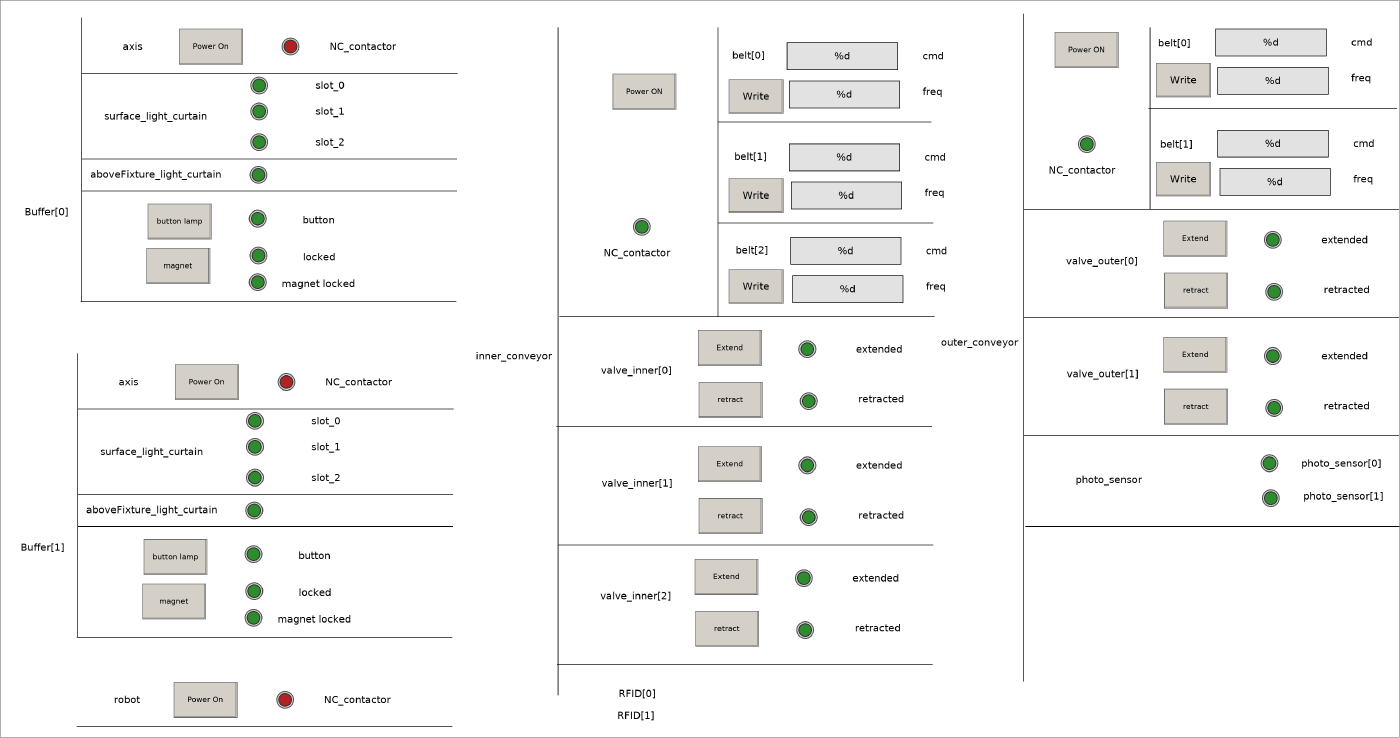
VISUALIZATION v_pm_0  // 2048x1080
VAR_IN_OUT
	dIO_PM		: Picking_Module;
END_VAR
    Lamp1 (364,110 30x30), variable: dIO_PM.buffer[0].surfae_slot_0, style: Lamp-Lamp1-Green
    Label (418,112 130x26), "slot_0"
    Label (28,297 80x26), "Buffer[0]"
    Line (120,107) (669,107)
    Line (119,26) (119,441)
    Line (118,441) (667,441)
    Label (672,508 160x26), "inner_conveyor"
    Line (816,40) (816,1017)
    Label (851,529 160x26), "valve_inner[0]"
    Button (1021,483 93x52), "Extend", colour toggle: dIO_PM.inConv.valve[0].extend
        OnMouseDown: execute { dIO_PM.inConv.valve[0].extend := TRUE; dIO_PM.inConv.valve[0].retract := FALSE; }
    Button (1022,559 93x52), "retract", colour toggle: dIO_PM.inConv.valve[0].retract
        OnMouseDown: execute { dIO_PM.inConv.valve[0].extend := FALSE; dIO_PM.inConv.valve[0].retract := TRUE; }
    Lamp1 (1166,496 30x30), variable: dIO_PM.inConv.valve[0].extended, style: Lamp-Lamp1-Green
    Lamp1 (1168,572 30x30), variable: dIO_PM.inConv.valve[0].retracted, style: Lamp-Lamp1-Green
    Label (1220,498 132x26), "extended"
    Label (1223,571 132x26), "retracted"
    Label (852,694 160x26), "valve_inner[1]"
    Label (850,859 160x26), "valve_inner[2]"
    Line (814,624) (1363,624)
    Line (816,797) (1365,797)
    Line (815,972) (1364,972)
    Label (465,55 132x26), "NC_contactor"
    Label (128,55 132x26), "axis"
    Button (262,42 93x52), "Power On", colour toggle: dIO_PM.buffer[0].power_axis
        toggle dIO_PM.buffer[0].power_axis
    Lamp1 (410,53 30x30), variable: dIO_PM.buffer[0].contractor_axis, style: Lamp-Lamp1-Red
    Label (128,157 200x26), "surface_light_curtain"
    Label (418,150 130x26), "slot_1"
    Lamp1 (364,148 30x30), variable: dIO_PM.buffer[0].surfae_slot_1, style: Lamp-Lamp1-Green
    Label (418,195 130x26), "slot_2"
    Lamp1 (364,193 30x30), variable: dIO_PM.buffer[0].surfae_slot_2, style: Lamp-Lamp1-Green
    Label (128,242 200x26), "aboveFixture_light_curtain"
    Lamp1 (363,241 30x30), variable: dIO_PM.buffer[0].above_fixture_light_curtain, style: Lamp-Lamp1-Green
    Line (119,232) (668,232)
    Line (119,279) (668,279)
    Label (406,309 120x26), "button"
    Lamp1 (362,305 30x30), variable: dIO_PM.buffer[0].button, style: Lamp-Lamp1-Green
    Button (216,298 93x52), "button lamp", colour toggle: dIO_PM.buffer[0].lamp_button
        toggle dIO_PM.buffer[0].lamp_button
    Button (214,363 93x52), "magnet", colour toggle: dIO_PM.buffer[0].magnet
        toggle dIO_PM.buffer[0].magnet
    Label (407,363 120x26), "locked"
    Lamp1 (363,359 30x30), variable: dIO_PM.buffer[0].locked, style: Lamp-Lamp1-Green
    Label (406,402 120x26), "magnet locked"
    Lamp1 (362,398 30x30), variable: dIO_PM.buffer[0].magnet_locked, style: Lamp-Lamp1-Green
    Lamp1 (358,601 30x30), variable: dIO_PM.buffer[1].surfae_slot_0, style: Lamp-Lamp1-Green
    Label (412,603 130x26), "slot_0"
    Label (22,788 80x26), "Buffer[1]"
    Line (114,598) (663,598)
    Line (113,517) (113,932)
    Line (112,932) (661,932)
    Label (459,546 132x26), "NC_contactor"
    Label (122,546 132x26), "axis"
    Button (256,533 93x52), "Power On", colour toggle: dIO_PM.buffer[1].power_axis
        toggle dIO_PM.buffer[1].power_axis
    Lamp1 (404,544 30x30), variable: dIO_PM.buffer[1].contractor_axis, style: Lamp-Lamp1-Red
    Label (122,648 200x26), "surface_light_curtain"
    Label (412,641 130x26), "slot_1"
    Lamp1 (358,639 30x30), variable: dIO_PM.buffer[1].surfae_slot_1, style: Lamp-Lamp1-Green
    Label (412,686 130x26), "slot_2"
    Lamp1 (358,684 30x30), variable: dIO_PM.buffer[1].surfae_slot_2, style: Lamp-Lamp1-Green
    Label (122,733 200x26), "aboveFixture_light_curtain"
    Lamp1 (357,732 30x30), variable: dIO_PM.buffer[1].above_fixture_light_curtain, style: Lamp-Lamp1-Green
    Line (113,723) (662,723)
    Line (113,770) (662,770)
    Label (400,800 120x26), "button"
    Lamp1 (356,796 30x30), variable: dIO_PM.buffer[1].button, style: Lamp-Lamp1-Green
    Button (210,789 93x52), "button lamp", colour toggle: dIO_PM.buffer[1].lamp_button
        toggle dIO_PM.buffer[1].lamp_button
    Button (208,854 93x52), "magnet", colour toggle: dIO_PM.buffer[1].magnet
        toggle dIO_PM.buffer[1].magnet
    Label (401,854 120x26), "locked"
    Lamp1 (357,850 30x30), variable: dIO_PM.buffer[1].locked, style: Lamp-Lamp1-Green
    Label (400,893 120x26), "magnet locked"
    Lamp1 (356,889 30x30), variable: dIO_PM.buffer[1].magnet_locked, style: Lamp-Lamp1-Green
    Line (112,1063) (661,1063)
    Label (457,1011 132x26), "NC_contactor"
    Label (120,1011 132x26), "robot"
    Button (254,998 93x52), "Power On", colour toggle: dIO_PM.power_robot
        toggle dIO_PM.power_robot
    Lamp1 (402,1009 30x30), variable: dIO_PM.contactor_robot, style: Lamp-Lamp1-Red
    Rectangle (1151,62 162x40), "%d", text variable: dIO_PM.inConv.belt[0].fbconverter.cmd
        OnMouseClick: write the text variable via Default
    Rectangle (1154,118 162x40), "%d", text variable: dIO_PM.inConv.belt[0].fbconverter.freq
        OnMouseClick: write the text variable via Default
    Label (1029,68 132x26), "belt[0]"
    Label (1299,69 132x26), "cmd"
    Label (1298,121 132x26), "freq"
    Line (1050,178) (1362,178)
    Rectangle (1154,210 162x40), "%d", text variable: dIO_PM.inConv.belt[1].fbconverter.cmd
        OnMouseClick: write the text variable via Default
    Rectangle (1157,266 162x40), "%d", text variable: dIO_PM.inConv.belt[1].fbconverter.freq
        OnMouseClick: write the text variable via Default
    Label (1032,216 132x26), "belt[1]"
    Label (1302,217 132x26), "cmd"
    Label (1301,269 132x26), "freq"
    Line (1050,326) (1365,326)
    Rectangle (1156,347 162x40), "%d", text variable: dIO_PM.inConv.belt[2].fbconverter.cmd
        OnMouseClick: write the text variable via Default
    Rectangle (1159,403 162x40), "%d", text variable: dIO_PM.inConv.belt[2].fbconverter.freq
        OnMouseClick: write the text variable via Default
    Label (1034,353 132x26), "belt[2]"
    Label (1304,354 132x26), "cmd"
    Label (1303,406 132x26), "freq"
    Line (818,463) (1367,463)
    Button (1021,653 93x52), "Extend", colour toggle: dIO_PM.inConv.valve[1].extend
        OnMouseDown: execute { dIO_PM.inConv.valve[1].extend := TRUE; dIO_PM.inConv.valve[1].retract := FALSE; }
    Button (1022,729 93x52), "retract", colour toggle: dIO_PM.inConv.valve[1].retract
        OnMouseDown: execute { dIO_PM.inConv.valve[1].extend := FALSE; dIO_PM.inConv.valve[1].retract := TRUE; }
    Lamp1 (1166,666 30x30), variable: dIO_PM.inConv.valve[1].extended, style: Lamp-Lamp1-Green
    Lamp1 (1168,742 30x30), variable: dIO_PM.inConv.valve[1].retracted, style: Lamp-Lamp1-Green
    Label (1220,668 132x26), "extended"
    Label (1223,741 132x26), "retracted"
    Button (1016,818 93x52), "Extend", colour toggle: dIO_PM.inConv.valve[2].extend
        OnMouseDown: execute { dIO_PM.inConv.valve[2].extend := TRUE; dIO_PM.inConv.valve[2].retract := FALSE; }
    Button (1017,894 93x52), "retract", colour toggle: dIO_PM.inConv.valve[2].retract
        OnMouseDown: execute { dIO_PM.inConv.valve[2].extend := FALSE; dIO_PM.inConv.valve[2].retract := TRUE; }
    Lamp1 (1161,831 30x30), variable: dIO_PM.inConv.valve[2].extended, style: Lamp-Lamp1-Green
    Lamp1 (1163,907 30x30), variable: dIO_PM.inConv.valve[2].retracted, style: Lamp-Lamp1-Green
    Label (1215,833 132x26), "extended"
    Label (1218,906 132x26), "retracted"
    Label (852,1002 160x26), "RFID[0]"
    Label (850,1034 160x26), "RFID[1]"
    Label (1353,488 160x26), "outer_conveyor"
    Line (1497,20) (1497,997)
    Label (1532,369 160x26), "valve_outer[0]"
    Button (1702,323 93x52), "Extend", colour toggle: dIO_PM.outConv.valve[0].extend
        OnMouseDown: execute { dIO_PM.outConv.valve[0].extend := TRUE; dIO_PM.outConv.valve[0].retract := FALSE; }
    Button (1703,399 93x52), "retract", colour toggle: dIO_PM.outConv.valve[0].retract
        OnMouseDown: execute { dIO_PM.outConv.valve[0].extend := FALSE; dIO_PM.outConv.valve[0].retract := TRUE; }
    Lamp1 (1847,336 30x30), variable: dIO_PM.outConv.valve[0].extended, style: Lamp-Lamp1-Green
    Lamp1 (1849,412 30x30), variable: dIO_PM.outConv.valve[0].retracted, style: Lamp-Lamp1-Green
    Label (1901,338 132x26), "extended"
    Label (1904,411 132x26), "retracted"
    Label (1533,534 160x26), "valve_outer[1]"
    Line (1498,464) (2047,464)
    Line (1497,637) (2046,637)
    Line (1500,770) (2049,770)
    Rectangle (1778,42 162x40), "%d", text variable: dIO_PM.outConv.belt[0].fbconverter.cmd
        OnMouseClick: write the text variable via Default
    Rectangle (1781,98 162x40), "%d", text variable: dIO_PM.outConv.belt[0].fbconverter.freq
        OnMouseClick: write the text variable via Default
    Label (1652,50 132x26), "belt[0]"
    Label (1926,49 132x26), "cmd"
    Label (1925,101 132x26), "freq"
    Line (1680,158) (2043,158)
    Rectangle (1781,190 162x40), "%d", text variable: dIO_PM.outConv.belt[1].fbconverter.cmd
        OnMouseClick: write the text variable via Default
    Rectangle (1784,246 162x40), "%d", text variable: dIO_PM.outConv.belt[1].fbconverter.freq
        OnMouseClick: write the text variable via Default
    Label (1655,198 132x26), "belt[1]"
    Label (1929,197 132x26), "cmd"
    Label (1928,249 132x26), "freq"
    Line (1497,306) (2046,306)
    Button (1702,493 93x52), "Extend", colour toggle: dIO_PM.outConv.valve[1].extend
        OnMouseDown: execute { dIO_PM.outConv.valve[1].extend := TRUE; dIO_PM.outConv.valve[1].retract := FALSE; }
    Button (1703,569 93x52), "retract", colour toggle: dIO_PM.outConv.valve[1].retract
        OnMouseDown: execute { dIO_PM.outConv.valve[1].extend := FALSE; dIO_PM.outConv.valve[1].retract := TRUE; }
    Lamp1 (1847,506 30x30), variable: dIO_PM.outConv.valve[1].extended, style: Lamp-Lamp1-Green
    Lamp1 (1849,582 30x30), variable: dIO_PM.outConv.valve[1].retracted, style: Lamp-Lamp1-Green
    Label (1901,508 132x26), "extended"
    Label (1904,581 132x26), "retracted"
    Lamp1 (1842,663 30x30), variable: dIO_PM.outConv.photo_sensor[0], style: Lamp-Lamp1-Green
    Lamp1 (1844,714 30x30), variable: dIO_PM.outConv.photo_sensor[1], style: Lamp-Lamp1-Green
    Label (1896,665 132x26), "photo_sensor[0]"
    Label (1899,713 132x26), "photo_sensor[1]"
    Label (1542,689 160x26), "photo_sensor"
    Line (1050,40) (1050,463)
    Button (896,108 93x52), "Power ON", colour toggle: dIO_PM.power_inConv
        toggle dIO_PM.power_inConv
    Lamp1 (924,317 30x30), variable: dIO_PM.contactor_inConv, style: Lamp-Lamp1-Green
    Label (866,357 132x26), "NC_contactor"
    Line (1682,40) (1682,306)
    Button (1543,47 93x52), "Power ON", colour toggle: dIO_PM.power_outConv
        toggle dIO_PM.power_outConv
    Lamp1 (1575,196 30x30), variable: dIO_PM.contactor_outConv, style: Lamp-Lamp1-Green
    Label (1517,236 132x26), "NC_contactor"
    Button (1066,116 80x50), "Write"
        OnMouseDown: execute { dIO_PM.inConv.belt[0].fbconverter.bSetParaEx	:= TRUE; }
        OnMouseUp: execute { dIO_PM.inConv.belt[0].fbconverter.bSetParaEx	:= FALSE; }
    Button (1066,261 80x50), "Write"
        OnMouseDown: execute { dIO_PM.inConv.belt[1].fbconverter.bSetParaEx	:= TRUE; }
        OnMouseUp: execute { dIO_PM.inConv.belt[1].fbconverter.bSetParaEx	:= FALSE; }
    Button (1066,394 80x50), "Write"
        OnMouseDown: execute { dIO_PM.inConv.belt[2].fbconverter.bSetParaEx	:= TRUE; }
        OnMouseUp: execute { dIO_PM.inConv.belt[2].fbconverter.bSetParaEx	:= FALSE; }
    Button (1691,237 80x50), "Write"
        OnMouseDown: execute { dIO_PM.outConv.belt[1].fbconverter.bSetParaEx	:= TRUE; }
        OnMouseUp: execute { dIO_PM.outConv.belt[1].fbconverter.bSetParaEx	:= FALSE; }
    Button (1691,92 80x50), "Write"
        OnMouseDown: execute { dIO_PM.outConv.belt[0].fbconverter.bSetParaEx	:= TRUE; }
        OnMouseUp: execute { dIO_PM.outConv.belt[0].fbconverter.bSetParaEx	:= FALSE; }
END_VISUALIZATION

(* stored: Version 1.1.0.1, ProductVersion 3.1.4024.12
   Visu v_pm_0: Id {578c3a9f-5229-4d6b-9d38-828533f2e485} *)
